TYPE E_CHM_WriteMode :
(
	E_CHM_FSS2MODE_NOBACKUP,
	E_CHM_FSS2MODE_FSS2BACKUP,
	E_CHM_FSS3MODE_NOBACKUP,
	E_CHM_FSS3MODE_FSS2BACKUP

);
END_TYPE

(* stored: Version 1.1.0.1, ProductVersion 3.1.4024.15
   DUT E_CHM_WriteMode: Id {c2bd096d-1f7c-4be6-b2ec-7830b1e93576} *)
